FUNCTION_BLOCK SifbCBPrintStatus
  (* Standard: 61499-2 *)
  (* Version 0.1, 2019-00-29, hpea485, UOA *)
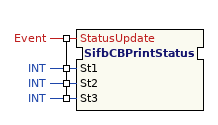
  EVENT_INPUT
    StatusUpdate WITH St1, St2, St3;
  END_EVENT
  VAR_INPUT
    St1 : INT;
    St2 : INT;
    St3 : INT;
  END_VAR
  VAR
    Variable1 : BOOL;
  END_VAR
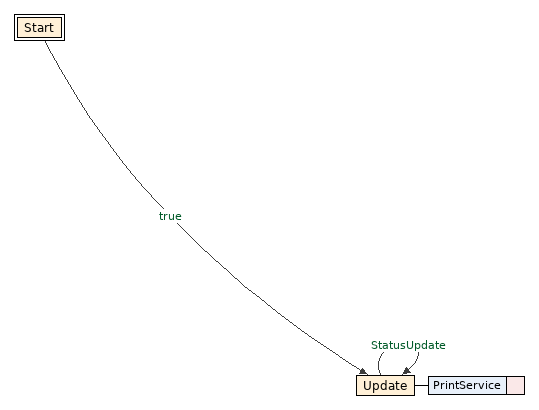
  EC_STATES
    Start;
    Update : PrintService;
  END_STATES
  EC_TRANSITIONS
    Start TO Update := true;
    Update TO Update := StatusUpdate;
  END_TRANSITIONS
  ALGORITHM PrintService IN C:
// OFF 0
// RUNNING 1
// WEIGHT -1
// LASER -2
// STALL -3
// SPEED -4

printf("CB 1: ");
switch(me->St1) {
	case 0:
		printf("CLOSED       ");
		break;
	case 1:
		printf("OPEN         ");
		break;
	default:
		printf("UNKNOWN      ");
		break;
}
printf("\t");

printf("CB 2: ");
switch(me->St1) {
	case 0:
		printf("CLOSED       ");
		break;
	case 1:
		printf("OPEN         ");
		break;
	default:
		printf("UNKNOWN      ");
		break;
}
printf("\t");

printf("CB 3: ");
switch(me->St1) {
	case 0:
		printf("CLOSED       ");
		break;
	case 1:
		printf("OPEN         ");
		break;
	default:
		printf("UNKNOWN      ");
		break;
}
printf("\n");
  END_ALGORITHM
END_FUNCTION_BLOCK
